// TIA Portal V18 export
// export: Created 2026-01-09T11:31:58.961875Z, ExportSetting WithDefaults, DisplayName Totally Integrated Automation Portal, DisplayVersion V18 Update 5, DisplayName TIA Portal Openness, DisplayVersion V18 Update 5, DisplayName TIA Portal Teamcenter Gateway, DisplayVersion V18, DisplayName TIA Portal Version Control Interface, DisplayVersion V18, DisplayName SINAMICS Startdrive Advanced, DisplayVersion V18 SP2 Update 1, DisplayName SINAMICS Startdrive G110M, G120, G120C, G120D, G120P, G115D, DisplayVersion V18 SP2 Update 1, DisplayName SINAMICS Startdrive G130, G150, S120, S150, SINAMICS MV, S210, G220, S200, DisplayVersion V18 SP2 Update 1, DisplayName STEP 7 Professional, DisplayVersion V18 Update 5, DisplayName STEP 7 Safety, DisplayVersion V18, DisplayName WinCC Professional, DisplayVersion V18 Update 5
TagTable "CylinderErrorWord"
  CylinderError1-4 : Word  (%DB1067.DBW0, CPU S71500-2PN_TP700, 100 ms)
  CylinderError5-8 : Word  (%DB1067.DBW2, CPU S71500-2PN_TP700, 100 ms)
  CylinderError9-12 : Word  (%DB1067.DBW4, CPU S71500-2PN_TP700, 100 ms)
  CylinderError13-16 : Word  (%DB1067.DBW6, CPU S71500-2PN_TP700, 100 ms)
  CylinderError17-20 : Word  (%DB1067.DBW8, CPU S71500-2PN_TP700, 100 ms)
  CylinderError21-24 : Word  (%DB1067.DBW10, CPU S71500-2PN_TP700, 100 ms)
  CylinderError25-28 : Word  (%DB1067.DBW12, CPU S71500-2PN_TP700, 100 ms)
  CylinderError29-32 : Word  (%DB1067.DBW14, CPU S71500-2PN_TP700, 100 ms)
  CylinderError33-36 : Word  (%DB1067.DBW16, CPU S71500-2PN_TP700, 100 ms)
  CylinderError37-40 : Word  (%DB1067.DBW18, CPU S71500-2PN_TP700, 100 ms)
  CylinderError41-44 : Word  (%DB1067.DBW20, CPU S71500-2PN_TP700, 100 ms)
  CylinderError45-48 : Word  (%DB1067.DBW22, CPU S71500-2PN_TP700, 100 ms)
  CylinderError49-52 : Word  (%DB1067.DBW24, CPU S71500-2PN_TP700, 100 ms)
  CylinderError53-56 : Word  (%DB1067.DBW26, CPU S71500-2PN_TP700, 100 ms)
  CylinderError57-60 : Word  (%DB1067.DBW28, CPU S71500-2PN_TP700, 100 ms)
  CylinderError61-64 : Word  (%DB1067.DBW30, CPU S71500-2PN_TP700, 100 ms)
  CylinderError65-68 : Word  (%DB1067.DBW32, CPU S71500-2PN_TP700, 100 ms)
  CylinderError69-72 : Word  (%DB1067.DBW34, CPU S71500-2PN_TP700, 100 ms)
  CylinderError73-76 : Word  (%DB1067.DBW36, CPU S71500-2PN_TP700, 100 ms)
  CylinderError77-80 : Word  (%DB1067.DBW38, CPU S71500-2PN_TP700, 100 ms)
  CylinderError81-84 : Word  (%DB1067.DBW40, CPU S71500-2PN_TP700, 100 ms)
  CylinderError85-88 : Word  (%DB1067.DBW42, CPU S71500-2PN_TP700, 100 ms)
  CylinderError89-92 : Word  (%DB1067.DBW44, CPU S71500-2PN_TP700, 100 ms)
  CylinderError93-96 : Word  (%DB1067.DBW46, CPU S71500-2PN_TP700, 100 ms)
  CylinderError97-100 : Word  (%DB1067.DBW48, CPU S71500-2PN_TP700, 100 ms)
  CylinderError101-104 : Word  (%DB1067.DBW50, CPU S71500-2PN_TP700, 100 ms)
  CylinderError105-108 : Word  (%DB1067.DBW52, CPU S71500-2PN_TP700, 100 ms)
  CylinderError109-112 : Word  (%DB1067.DBW54, CPU S71500-2PN_TP700, 100 ms)
  CylinderError113-116 : Word  (%DB1067.DBW56, CPU S71500-2PN_TP700, 100 ms)
  CylinderError117-120 : Word  (%DB1067.DBW58, CPU S71500-2PN_TP700, 100 ms)
  CylinderError121-124 : Word  (%DB1067.DBW60, CPU S71500-2PN_TP700, 100 ms)
  CylinderError125-128 : Word  (%DB1067.DBW62, CPU S71500-2PN_TP700, 100 ms)
  CylinderError129-132 : Word  (%DB1067.DBW64, CPU S71500-2PN_TP700, 100 ms)
  CylinderError133-136 : Word  (%DB1067.DBW66, CPU S71500-2PN_TP700, 100 ms)
  CylinderError137-140 : Word  (%DB1067.DBW68, CPU S71500-2PN_TP700, 100 ms)
  CylinderError141-144 : Word  (%DB1067.DBW70, CPU S71500-2PN_TP700, 100 ms)
  CylinderError145-148 : Word  (%DB1067.DBW72, CPU S71500-2PN_TP700, 100 ms)
  CylinderError149-152 : Word  (%DB1067.DBW74, CPU S71500-2PN_TP700, 100 ms)
  CylinderError153-156 : Word  (%DB1067.DBW76, CPU S71500-2PN_TP700, 100 ms)
  CylinderError157-160 : Word  (%DB1067.DBW78, CPU S71500-2PN_TP700, 100 ms)
  CylinderError161-164 : Word  (%DB1067.DBW80, CPU S71500-2PN_TP700, 100 ms)
  CylinderError165-168 : Word  (%DB1067.DBW82, CPU S71500-2PN_TP700, 100 ms)
  CylinderError169-172 : Word  (%DB1067.DBW84, CPU S71500-2PN_TP700, 100 ms)
  CylinderError173-176 : Word  (%DB1067.DBW86, CPU S71500-2PN_TP700, 100 ms)
  CylinderError177-180 : Word  (%DB1067.DBW88, CPU S71500-2PN_TP700, 100 ms)
  CylinderError181-184 : Word  (%DB1067.DBW90, CPU S71500-2PN_TP700, 100 ms)
  CylinderError185-188 : Word  (%DB1067.DBW92, CPU S71500-2PN_TP700, 100 ms)
  CylinderError189-192 : Word  (%DB1067.DBW94, CPU S71500-2PN_TP700, 100 ms)
  CylinderError193-196 : Word  (%DB1067.DBW96, CPU S71500-2PN_TP700, 100 ms)
  CylinderError197-200 : Word  (%DB1067.DBW98, CPU S71500-2PN_TP700, 100 ms)
